PROGRAM P_Demo_FB_HVACSetpointHeating
VAR
    fb : FB_HVACSetpointHeating;                            // 被演示 FB 实例
    eDataSecurityType_in : E_HVACDataSecurityType ;
    bSetDefault_in : BOOL := FALSE;
    bEnable_in : BOOL := FALSE;
    rSetpointIn_in : REAL := 0.0;
    rOutsideTempDamped_in : REAL := 0.0;
    dtSystemTime_in : DT ;
    bDayOperation_in : BOOL := FALSE;
    bFreezeProtec_in : BOOL := FALSE;
    bReset_in : BOOL := FALSE;
    rSetpointOut_out : REAL;
    bHeating_out : BOOL;
    bReqOutsideTemp_out : BOOL;
    bReqDate_out : BOOL;
    bReqPermanent_out : BOOL;
    bReqFreezeProtec_out : BOOL;
    bReqNight_out : BOOL;
    bReqDay_out : BOOL;
    bInvalidParameter_out : BOOL;
END_VAR

// ============================================================================
// Tc2_HVAC.FB_HVACSetpointHeating 演示程序
// ============================================================================
// 场景：把本 FB 实例化到一个 PLC 程序里，每周期单次调用；按需要把 VAR_INPUT 与
//       VAR_IN_OUT 接到工程信号；VAR_OUTPUT 写入对应监视变量。
// 价值：使用本 FB 比手写状态机 / 控制算法节省大量代码；与 Tc2_HVAC 体系内其它 FB
//       直接对接，命名 / 持久化 / 模式仲裁等约定一致。具体语义见 FB_HVACSetpointHeating.md 主文档。
// 验证步骤：
//   1. 右键 PLC 项目下 POUs 文件夹 → Add → Existing Item → 选本 .TcPOU 文件
//   2. 引用 Tc2_HVAC（References → Add library）
//   3. 编译 → 登录 → 运行
//   4. 在线写各 *_in 输入信号触发 FB；在线 monitor *_out 引脚观察状态
// ============================================================================

fb(
    eDataSecurityType := eDataSecurityType_in,
    bSetDefault := bSetDefault_in,
    bEnable := bEnable_in,
    rSetpointIn := rSetpointIn_in,
    rOutsideTempDamped := rOutsideTempDamped_in,
    dtSystemTime := dtSystemTime_in,
    bDayOperation := bDayOperation_in,
    bFreezeProtec := bFreezeProtec_in,
    bReset := bReset_in,
    rSetpointOut => rSetpointOut_out,
    bHeating => bHeating_out,
    bReqOutsideTemp => bReqOutsideTemp_out,
    bReqDate => bReqDate_out,
    bReqPermanent => bReqPermanent_out,
    bReqFreezeProtec => bReqFreezeProtec_out,
    bReqNight => bReqNight_out,
    bReqDay => bReqDay_out,
    bInvalidParameter => bInvalidParameter_out
);

END_PROGRAM

(* stored: Version 1.1.0.1, ProductVersion 3.1.4024.5
   POU P_Demo_FB_HVACSetpointHeating: Id {7dbb9f98-7a6f-5c17-bbbe-1d763229fad4}, SpecialFunc None *)
